// TIA Portal V19 export
FUNCTION "Ax_PB_Connector" : Void   // FC156, LAD
TITLE = Collect push buttons for Axis machines
// stored: Access Published, SetENOAutomatically false
   VAR_INPUT
      Enable : Bool;
      HMI_PB : "Ax_PB";   // Push button from HMI a (e.g. MB1)
      LB_PB_Bwd_Minus : Bool;
      LB_PB_Fwd_Plus : Bool;
      LB_PB_MoveToPos : Bool;
      Other_PB : "Ax_PB";
   END_VAR
   VAR_OUTPUT
      PB : "Ax_PB";   // Push button from HMI a (e.g. MB1)
   END_VAR
BEGIN

REGION Network 1: Logical OR
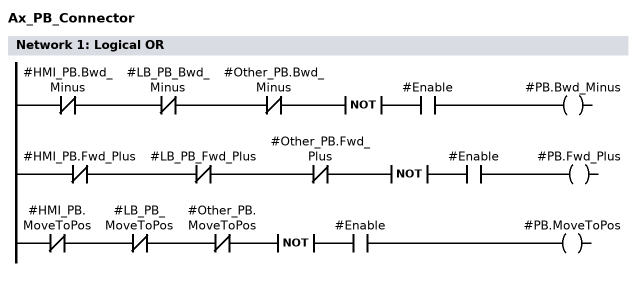
   RUNG wire#powerrail
      I_Contact( #HMI_PB.Bwd_Minus )
      I_Contact( #LB_PB_Bwd_Minus )
      I_Contact( #Other_PB.Bwd_Minus )
      Not()
      Contact( #Enable )
      Coil( #PB.Bwd_Minus )
   END_RUNG
   RUNG wire#powerrail
      I_Contact( #HMI_PB.Fwd_Plus )
      I_Contact( #LB_PB_Fwd_Plus )
      I_Contact( #Other_PB.Fwd_Plus )
      Not()
      Contact( #Enable )
      Coil( #PB.Fwd_Plus )
   END_RUNG
   RUNG wire#powerrail
      I_Contact( #HMI_PB.MoveToPos )
      I_Contact( #LB_PB_MoveToPos )
      I_Contact( #Other_PB.MoveToPos )
      Not()
      Contact( #Enable )
      Coil( #PB.MoveToPos )
   END_RUNG
   // the same network as SCL:
   #PB.Bwd_Minus := NOT (NOT #HMI_PB.Bwd_Minus AND NOT #LB_PB_Bwd_Minus AND NOT #Other_PB.Bwd_Minus) AND #Enable;
   #PB.Fwd_Plus := NOT (NOT #HMI_PB.Fwd_Plus AND NOT #LB_PB_Fwd_Plus AND NOT #Other_PB.Fwd_Plus) AND #Enable;
   #PB.MoveToPos := NOT (NOT #HMI_PB.MoveToPos AND NOT #LB_PB_MoveToPos AND NOT #Other_PB.MoveToPos) AND #Enable;
END_REGION
END_FUNCTION
